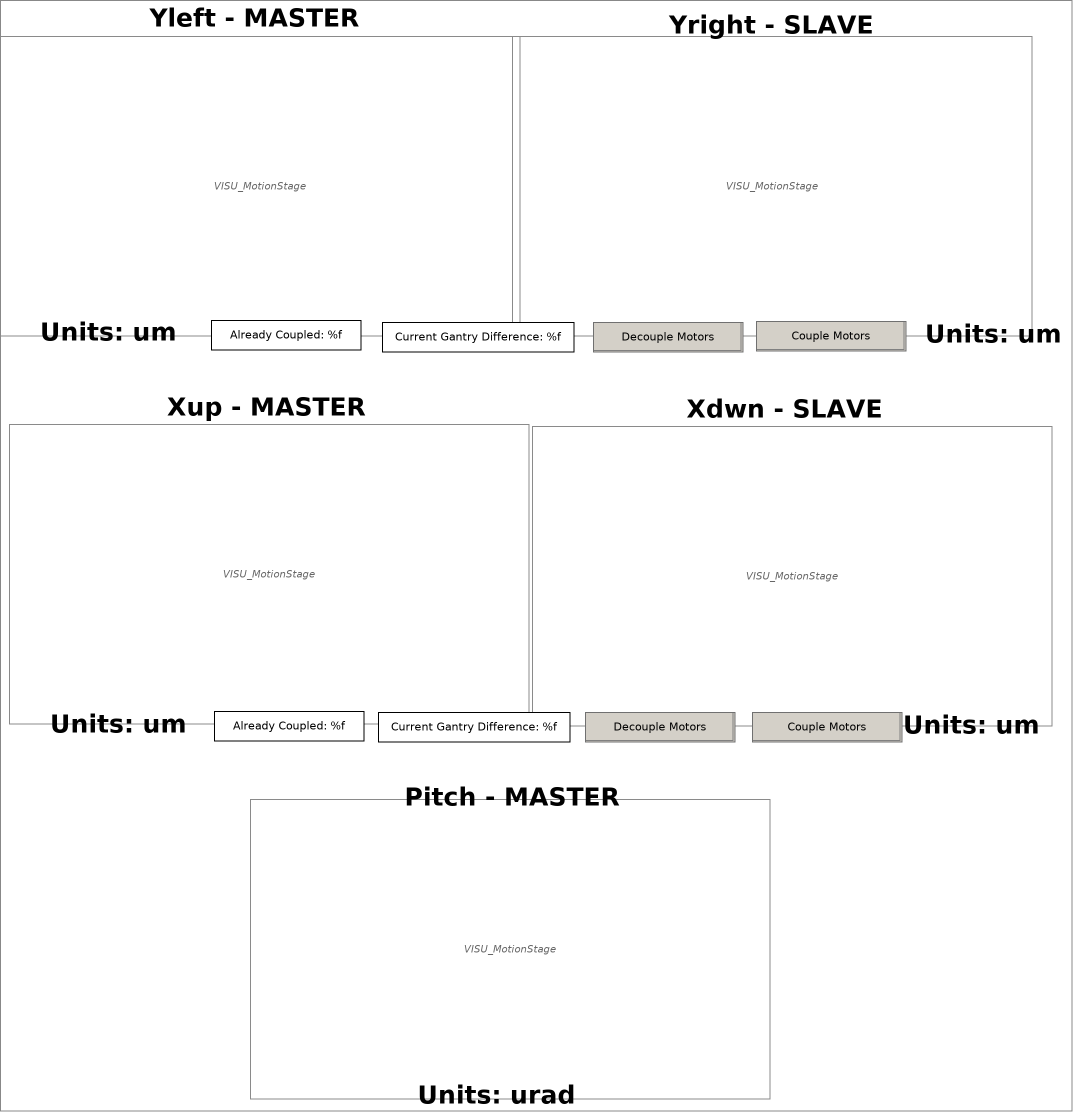
VISUALIZATION Visualization  // 1073x1112
    Label (14,2 481x31), "Yleft - MASTER"
    Frame (0,36 520x300)
        shows VISU_MotionStage(VisuMotionStage := MAIN.M1, Extras := MAIN.M1_Extras)
    Frame (512,36 520x300)
        shows VISU_MotionStage(VisuMotionStage := MAIN.M2, Extras := MAIN.M2_Extras)
    Label (531,9 481x31), "Yright - SLAVE"
    Rectangle (211,320 150x30), "Already Coupled: %f", tooltip "Couple Status: TRUE if coupled", text variable: MAIN.bGantryAlreadyCoupledY
    Rectangle (382,322 192x30), "Current Gantry Difference: %f", tooltip "Current Gantry Difference in um", text variable: MAIN.fCurrGantryY_um
    Button (593,322 150x30), "Decouple Motors", tooltip "Press To Decouple Motors for independent control", colour toggle: MAIN.bExecuteDecoupleY
    Button (756,321 150x30), "Couple Motors", tooltip "Press To Couple Motors", colour toggle: MAIN.bExecuteCoupleY
    Frame (9,424 520x300)
        shows VISU_MotionStage(VisuMotionStage := MAIN.M3, Extras := MAIN.M3_Extras)
    Label (26,391 481x31), "Xup - MASTER"
    Frame (532,426 520x300)
        shows VISU_MotionStage(VisuMotionStage := MAIN.M4, Extras := MAIN.M4_Extras)
    Label (544,393 481x31), "Xdwn - SLAVE"
    Rectangle (214,711 150x30), "Already Coupled: %f", tooltip "Couple Status: TRUE if coupled", text variable: MAIN.bGantryAlreadyCoupledX
    Rectangle (378,712 192x30), "Current Gantry Difference: %f", tooltip "Current Gantry Difference in um", text variable: MAIN.fCurrGantryX_um
    Button (585,712 150x30), "Decouple Motors", tooltip "Press To Decouple Motors for independent control", colour toggle: MAIN.bExecuteDecoupleX
    Button (752,712 150x30), "Couple Motors", tooltip "Press To Couple Motors", colour toggle: MAIN.bExecuteCoupleX
    Frame (250,799 520x300)
        shows VISU_MotionStage(VisuMotionStage := MAIN.M5, Extras := MAIN.M5_Extras)
    Label (272,781 481x31), "Pitch - MASTER"
    Label (31,316 155x31), "Units: um"
    Label (916,318 155x31), "Units: um"
    Label (41,708 155x31), "Units: um"
    Label (894,709 155x31), "Units: um"
    Label (419,1079 155x31), "Units: urad"
END_VISUALIZATION

(* stored: Version 1.1.0.1, ProductVersion 3.1.4022.18
   Visu Visualization: Id {af2f16f4-e7e7-4019-a84a-cc323e4115d2} *)
